FUNCTION_BLOCK BACnetBinaryInput (* Service Interface Function Block Type *)
  (* Standard: 61499-2 *)
  (* Version 1.0, 2020-03-03, root *)
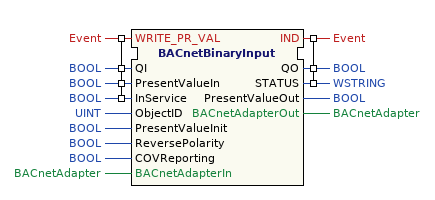
  EVENT_INPUT
    WRITE_PR_VAL WITH PresentValueIn, QI, InService; (* Write Present_Value event *)
  END_EVENT
  EVENT_OUTPUT
    IND WITH QO, STATUS; (* Present_Value write indication *)
  END_EVENT
  VAR_INPUT
    QI : BOOL; (* Event Input Qualifier *)
    PresentValueIn : BOOL; (* Value to be written into the Present_Value property *)
    InService : BOOL; (* Lifestatus flag of the object *)
    ObjectID : UINT; (* Identifier of the object *)
    PresentValueInit : BOOL; (* Initial value of the Present_Value property *)
    ReversePolarity : BOOL; (* Enable/Disable reverse polarity flag *)
    COVReporting : BOOL; (* Enable/Disable COV reporting flag *)
  END_VAR
  VAR_OUTPUT
    QO : BOOL; (* Event Output Qualifier *)
    STATUS : WSTRING; (* Status *)
    PresentValueOut : BOOL; (* Value of the Present_Value property *)
  END_VAR
  SOCKETS
    BACnetAdapterIn : BACnetAdapter; (* BACnet adapter socket *)
  END_SOCKETS
  PLUGS
    BACnetAdapterOut : BACnetAdapter; (* BACnet adapter plug *)
  END_PLUGS
END_FUNCTION_BLOCK
